// TIA Portal V16 export
// export: Created 2021-11-12T13:32:37.4172055Z, ExportSetting WithDefaults, DisplayName Totally Integrated Automation Portal, DisplayVersion V16 Update 3, DisplayName TIA Portal Version Control Interface, DisplayVersion V16 Update 2, DisplayName TIA Portal Openness, DisplayVersion V16 Update 3, DisplayName SINAMICS Startdrive Advanced, DisplayVersion V16 Update 5, DisplayName SINAMICS Startdrive G130, G150, S120, S150, SINAMICS MV, S210, DisplayVersion V16 Update 5, DisplayName SINAMICS Startdrive G110M, G120, G120C, G120D, G120P, G115D, DisplayVersion V16 Update 5, DisplayName STEP 7 Professional, DisplayVersion V16 Update 3, DisplayName STEP 7 Safety, DisplayVersion V16, DisplayName WinCC UA Professional, DisplayVersion V16 Update 3
DATA_BLOCK "IDB_Station230"   // DB37
VERSION : 0.1
// stored: AutoNumber true, DBAccessibleFromOPCUA true, InstanceOfName Station230, InstanceOfType FB
"Station230"
   // VAR
   //    SF_CL01_Alarm { S7_SetPoint := 'True'} : "STD_DI_Mon";
   //    SF_CL01_Warning { S7_SetPoint := 'True'} : "STD_DI_Mon";
   //    SF_GL01MA01 { S7_SetPoint := 'True'} : "STD_Drive1";
   //    SF_UC12TA01 { S7_SetPoint := 'True'} : "STD_Siemens_G120_CU240E_2_PN";
   //    SF_GL02MA01 { S7_SetPoint := 'True'} : "STD_Drive1";
   //    SF_UC12TA02 { S7_SetPoint := 'True'} : "STD_Siemens_G120_CU240E_2_PN";
   //    SF_TON_1 { S7_SetPoint := 'True'} : TON_TIME;
   //    SF_TOF_1 { S7_SetPoint := 'True'} : TOF_TIME;
   //    SF_CL01 { S7_SetPoint := 'True'} : "STD_PartCounter";
   //    SS_Edge { S7_SetPoint := 'True'} : Array[0..15] of Bool;
   //    SB1BoxExchangeReq { S7_SetPoint := 'True'} : Bool;
   // END_VAR
BEGIN
END_DATA_BLOCK
